// TIA Portal V20 export
TYPE "LBP_typeInternal1"
TITLE = Internal data type for basic program / Type de données interne pour programme de base
// Data type only for internal use in the basic program / Type de données réservé à l'utilisation interne dans le programme de base
   STRUCT
      active : Bool;
      mcpAddress : USInt;
      modeDCK : Bool;
      clientPort : UInt;
      connectionId : CONN_OUC;
      mcpClientReference : Word;
      mcpInPointer : Struct
         DbNumber : Word;
         PointerAddress : DWord;
      END_STRUCT;
      mcpOutPointer : Struct
         DbNumber : Word;
         PointerAddress : DWord;
      END_STRUCT;
      mcpDefaultInLength : UInt;
      mcpDefaultOutLength : UInt;
      useIpAddress : Bool;
      ipAddress : Array[1..4] of USInt;
   END_STRUCT;
END_TYPE
